TYPE ST_PointTestData :
STRUCT
//	udnPointNum		: UDINT;
	lrPosition 		: LREAL;
//	tTimeToPosition : TIME;
//	lrDistance		: LREAL;
	lrInitialVelo	: LREAL;
//	lrAvgVelo		: LREAL;
	lrFinalVelo		: LREAL;
	lrAccelDecel	: LREAL;
//	tTimeExecuted	: TIME;
//	lrFinalVeloActual	: LREAL;
	sMoveType		: STRING;
END_STRUCT
END_TYPE

(* stored: Version 1.1.0.1, ProductVersion 3.1.4022.3
   DUT ST_PointTestData: Id {085b5b6c-c90a-46be-bf8d-2a40463b6234} *)
